// Mitsubishi GX Works2 project: 시퀀스 예제 1   PLC: Q03UDV

PROGRAM MAIN
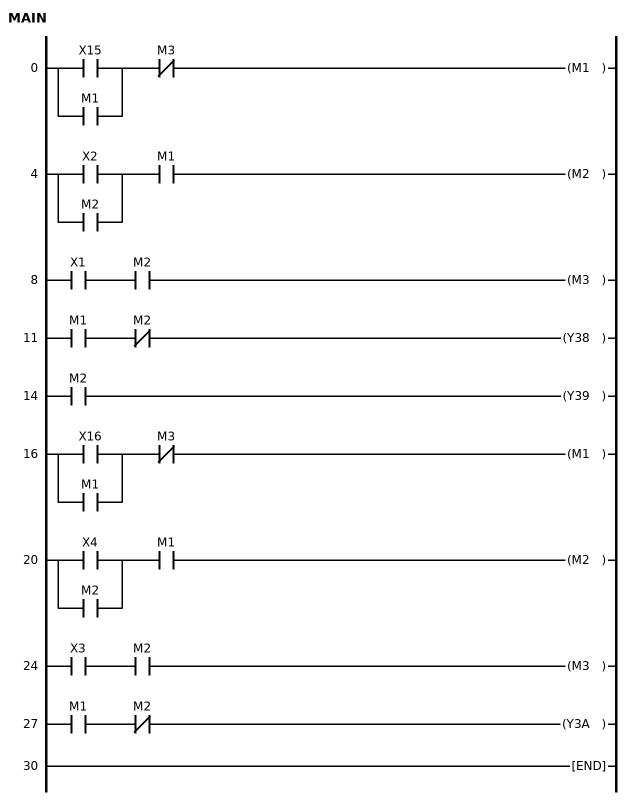
0     LD      X15
      OR      M1
      ANI     M3
      OUT     M1
4     LD      X2
      OR      M2
      AND     M1
      OUT     M2
8     LD      X1
      AND     M2
      OUT     M3
11    LD      M1
      ANI     M2
      OUT     Y38
14    LD      M2
      OUT     Y39
16    LD      X16
      OR      M1
      ANI     M3
      OUT     M1
20    LD      X4
      OR      M2
      AND     M1
      OUT     M2
24    LD      X3
      AND     M2
      OUT     M3
27    LD      M1
      ANI     M2
      OUT     Y3A
30    END
END_PROGRAM
